INTERFACE I_SynchronousRpcHandlers

PROPERTY PUBLIC HasHandlers : BOOL
GET
END_GET
END_PROPERTY

METHOD PUBLIC TryGetByMethodName : BOOL
VAR_INPUT
	MethodName : T_MAXSTRING;
	Destination : REFERENCE TO I_SynchronousRpcHandler;
END_VAR
END_METHOD

END_INTERFACE

(* stored: Version 1.1.0.1, ProductVersion 3.1.4026.13
   Itf I_SynchronousRpcHandlers: Id {17486ac8-f2d6-46cc-89b1-d5123a0f9079}
   Property HasHandlers: Id {6d5593a1-560d-0ad7-3fd8-29e2e8670135}
   Get Get: Id {5006c248-002a-0111-28a5-03d992df5e5d}
   Method TryGetByMethodName: Id {29d8acf6-ba77-4e7a-86fb-b094662f8cf1} *)
